{attribute 'GeneratedUsingTerminal: KL9900-0063'}
{attribute addProperty BoxType "KL9900-0063"}
{attribute addProperty Id "Key_1AT %I*BOOL0Key_2AT %I*BOOL0Key_3AT %I*BOOL0Input_1AT %I*BOOL0Input_2AT %I*BOOL0Input_3AT %I*BOOL0LED_1AT %Q*BOOL0LED_2AT %Q*BOOL0LED_3AT %Q*BOOL0"}
{attribute addProperty CRC "1824580134"}
{attribute addProperty Size "0"}
TYPE Channel_6CC0E226 :
STRUCT
	{attribute addProperty Name "Key_1"}
	Key_1 AT %I* : BOOL;
	{attribute addProperty Name "Key_2"}
	Key_2 AT %I* : BOOL;
	{attribute addProperty Name "Key_3"}
	Key_3 AT %I* : BOOL;
	{attribute addProperty Name "Input_1"}
	Input_1 AT %I* : BOOL;
	{attribute addProperty Name "Input_2"}
	Input_2 AT %I* : BOOL;
	{attribute addProperty Name "Input_3"}
	Input_3 AT %I* : BOOL;
	{attribute addProperty Name "LED_1"}
	LED_1 AT %Q* : BOOL;
	{attribute addProperty Name "LED_2"}
	LED_2 AT %Q* : BOOL;
	{attribute addProperty Name "LED_3"}
	LED_3 AT %Q* : BOOL;
END_STRUCT
END_TYPE

(* stored: Version 1.2.0.0, ProductVersion 3.1.4024.9
   DUT Channel_6CC0E226: Id {b6a7e820-8d6e-4a05-9e99-7af20dcb735c} *)
